RoboDK station: UR3_automated.rdk

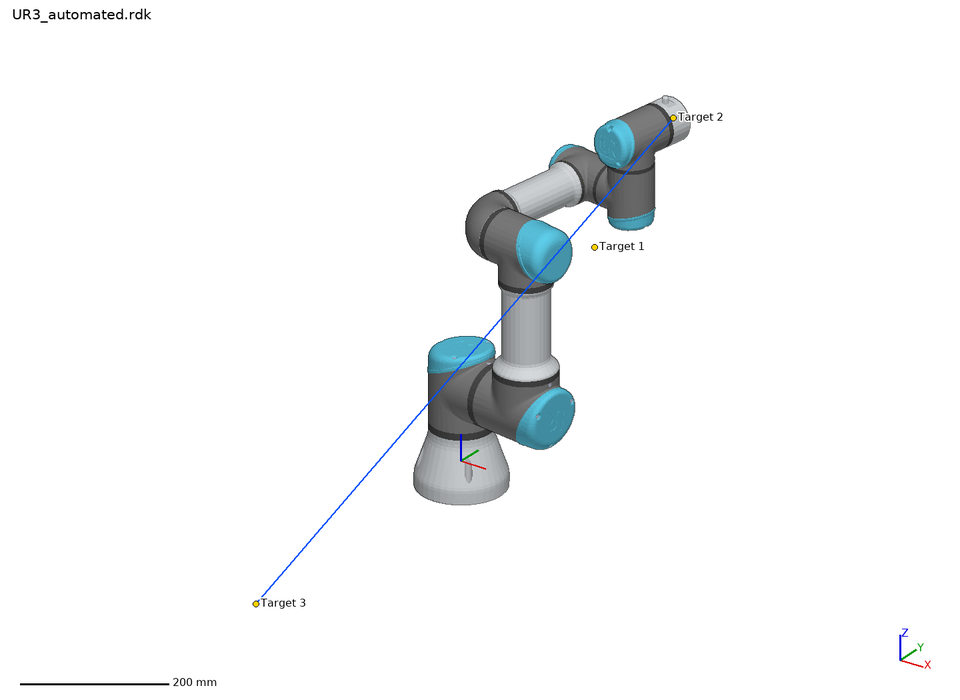
[picture v0: the station drawn from its stored meshes, robots at their saved joint values, targets as dots, program paths as lines]
Station UR3_automated. Poses are relative to the parent item; angles as X-Y-Z fixed-axis rotations.
  - frame UR3 Base at (0, 0, 0) mm
    - robot UR3: 6 axes, payload 3 kg, reach 500 mm, repeatability 0.1 mm, weight 11 kg
        modified DH rows (alpha deg, a mm, theta deg, d mm): 0, 0, 0, 118; 90, 0, 180, 0; 0, 243.65, 0, 0; 0, 213, 0, 110.4; -90, 0, 0, 83.4; 90, 0, 180, 82.4
        joint limits [-360, -360, -360, -360, -360, -360] to [360, 360, 360, 360, 360, 360]; home [0, -90, -90, 0, 90, 0]; saved at [81.14, -90, -90, 0, 90, 0]
    - target Target 1 (Cartesian target) at (295.4, -110.4, 445.05) mm, rotated rx -90 ry 0 rz -90 deg; joints [0, -90, -90, 0, 90, 0] of UR3
    - target Target 2 (Cartesian target) at (154.58, 274.87, 445.05) mm, rotated rx -90 ry 0 rz -8.86 deg; joints [81.14, -90, -90, 0, 90, 0] of UR3
    - target Target 3 (Cartesian target) at (30.25, -522.73, 4.08) mm, rotated rx 106.05 ry 0 rz -8.86 deg; joints [81.14, 4.59, -6.88, 18.34, 90, 0] of UR3
  - Python program Prog1 (listed below)
  - program Prog2 (2 instructions, listed below)
  - program Prog3 (3 instructions, listed below)
  - Python program Prog4 (listed below)
  - object Curve:R475;X-450;D50;A5 at (0, 0, 0) mm
  - object Curve:R475;X-450;D50;A5 at (0, 0, 0) mm
  - object Curve at (0, 0, 0) mm
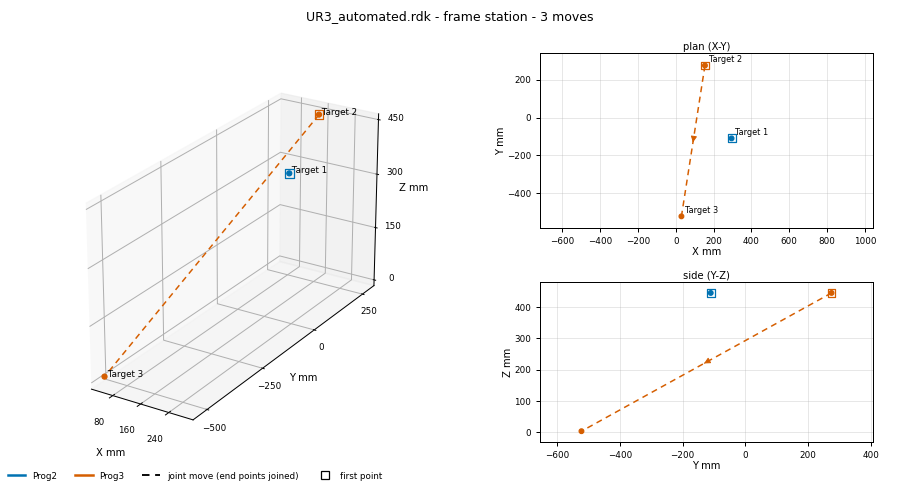
[picture p0: tool path of UR3_automated.rdk in frame station, 3 of 3 moves have a stored position in this frame; points joined in program order, loops and branches not executed]

--- Python program Prog1 ---
# Type help("robolink") or help("robodk") for more information
# Press F5 to run the script
# Documentation: https://robodk.com/doc/en/RoboDK-API.html
# Reference:     https://robodk.com/doc/en/PythonAPI/index.html
# Note: It is not required to keep a copy of this file, your python script is saved with the station
from robolink import *    # RoboDK's API
from robodk import *      # Math toolbox for robots

# Start the RoboDK API:
RDK = Robolink()

# Get the robot item by name:
robot = RDK.Item('UR3', ITEM_TYPE_ROBOT)

# Get the reference target by name:
R = 100

for i in range(2):
    target = RDK.Item('Target %s' % (i+1))
    target_pose = target.Pose()
    xyz_ref = target_pose.Pos()

    # Move the robot to the reference point:
    robot.MoveJ(target)
    # Draw a hexagon around the reference target:
    for i in range(7):
        ang = i * 2 * pi / 6 # ang = 0, 60, 120, ..., 360

        # Calculate the new position around the reference:
        x = xyz_ref[0] + R * cos(ang) # new X coordinate
        y = xyz_ref[1] + R * sin(ang) # new Y coordinate
        z = xyz_ref[2]                # new Z coordinate
        target_pose.setPos([x,y,z])

        # Move to the new target:
        robot.MoveL(target_pose)

    # Trigger a program call at the end of the movement
    # robot.RunCode('Program_Done')

# Move back to the reference target:
robot.MoveL(target)

--- program Prog2 (robot UR3) ---
  Set Ref.: UR3 Base
  MoveJ (Target 1)

--- program Prog3 (robot UR3) ---
  Set Ref.: UR3 Base
  MoveJ (Target 2)
  MoveJ (Target 3)

--- Python program Prog4 ---
# Type help("robolink") or help("robodk") for more information
# Press F5 to run the script

# This script shows an example of how a path curve can be added to a RoboDK station.
# The curve can be optionally projected to an existing object (either along the curve normals or to the closes distance)
#
# projection types (for AddCurve, as defined in robolink.py):
#PROJECTION_NONE                = 0 # No curve projection
#PROJECTION_CLOSEST             = 1 # The projection will the closest point on the surface
#PROJECTION_ALONG_NORMAL        = 2 # The projection will be done along the normal.
#PROJECTION_ALONG_NORMAL_RECALC = 3 # The projection will be done along the normal. Furthermore, the normal will be recalculated according to the surface normal.
# More information about the RoboDK API here:
# https://robodk.com/doc/en/RoboDK-API.html

# Function definition to create a list of points (curve)
def CirclePoints(radius, xStart, xEnd, xStep, accuracy, ycoord, projection):
    """Generates a list of points given circle dimensions"""
    nx,ny,nz = projection # normal/projection direction
    # Safe checks:
    radius = abs(radius)
    xStep = abs(xStep)
    accuracy = abs(accuracy)
    if abs(xStart) >= radius:
        raise Exception("Start point is outside the circle")
    if abs(xEnd) >= radius:
        raise Exception("End point is outside the circle")
    if xStart > xEnd:
        xStep = -xStep

    # Iterate on X coordinate, then on Z coordinate
    POINTS = []
    zSense = +1.0
    x = xStart
    x_steps = int(abs((xEnd - xStart)/xStep))
    y = ycoord
    for i in range(x_steps+1):
        z_abs = sqrt(radius*radius - x*x)
        z_steps = int(2*z_abs/accuracy)
        z_step = -zSense*2*z_abs/z_steps
        z = zSense*z_abs
        for j in range(z_steps+1):
            point_i = [x,y,z,nx,ny,nz] # create a ne point with normal/projection direction
            POINTS.append(point_i)
            z = z + z_step
        zSense = zSense * (-1.0)
        x = x + xStep
    return POINTS

#------------------------------------------------------------------
#--------------- PROGRAM START ---------------------
from robolink import *    # API to communicate with RoboDK
from robodk import *      # basic matrix operations

# Default parameters:
RADIUS = 475   # Radius of the outer circle
xSTART = -450  # Start point for the zig-zag
xEND   = 450   # End point for the zig-zag
xSTEP  = 50    # Step between passes
ACCURACY = 5   # Accuracy to cut the passes

# Other parameters:
yLEVEL = 200 # y coordinate, to start projection
proj_dir = [0,1,0] # projection direction -> normal/direction of the projection


# Initialize the RoboDK API
RDK = Robolink()

# Ask the user to select an object to project the curve
obj = RDK.ItemUserPick('Select object to project the path<br>(select cancel if you do not want to project the path)', ITEM_TYPE_OBJECT)

# Show message to the user
text = mbox("Enter the path parameters. Example:\n[RADIUS  xSTART  xEND  xSTEP  ACCURACY]", entry="475  -450  450  50  5")
if text:
    print("User entered:")
    print(text)
    # if the user entered the values, retrieve the list of values
    numbers = [float(x) for x in text.split()] # convert strings to numbers
    if len(numbers) >= 5:
        RADIUS, xSTART, xEND, xSTEP, ACCURACY = numbers # split array into variables
    else:
        print("Using default parameters")

else:
    print("Using default parameters")

# Generate the curve path
CURVE = CirclePoints(RADIUS, xSTART, xEND, xSTEP, ACCURACY, yLEVEL, proj_dir)

# display the points
print(CURVE)

# Add the curve to the object with the option to project along the normals and recalculate the normals according to the surface normal
curve = obj.AddCurve(CURVE, False, PROJECTION_ALONG_NORMAL_RECALC)
# last call is equivalent to:
RDK.AddCurve(CURVE, obj, False, PROJECTION_ALONG_NORMAL_RECALC)

curve.setName('Curve:R%.0f;X%.0f;D%.0f;A%.0f' % (RADIUS, xSTART, xSTEP, ACCURACY))
